PROGRAM MAIN
VAR
	Profiler: PROFILER;
	ProfilerResult  : PROFILERSTRUCT;
	nFactorial: ULINT;
END_VAR

Profiler(START:=TRUE,RESET:=TRUE);
Factorial(n:=nFactorial);
Profiler(START:=FALSE);
ProfilerResult:= Profiler.Data;

END_PROGRAM

(* stored: Version 1.1.0.1, ProductVersion 3.1.4024.12
   POU MAIN: Id {8b3f2565-88f1-4b08-803e-118186d0112d}, SpecialFunc None *)
